TYPE UValues :
UNION
	Binary: BOOL;
	Numeric: LREAL;
	String_t: STRING;
END_UNION
END_TYPE

(* stored: Version 1.1.0.1
   DUT UValues: Id {dac0e663-626c-40ef-a7b3-03281dab3016} *)
